FUNCTION_BLOCK FB_VeggiePizza EXTENDS FB_Pizza
VAR_INPUT
END_VAR
VAR_OUTPUT
END_VAR
VAR
END_VAR

METHOD addCheese
VAR_INPUT
END_VAR
ADSLOGSTR( msgCtrlMask := ADSLOG_MSGTYPE_WARN,
        	msgFmtStr := 'Adding Mozzarella Cheese...', '');
END_METHOD

METHOD addMeat
VAR_INPUT
END_VAR
// Nothing here because it's not used
// Normally these Meat, Cheese, and Veg would be an Abstract Method
END_METHOD

METHOD addVegetables : BOOL
VAR_INPUT
END_VAR
ADSLOGSTR( msgCtrlMask := ADSLOG_MSGTYPE_WARN,
        	msgFmtStr := 'Adding Veggies...', '');
END_METHOD

METHOD customerWantsCheese : BOOL
VAR_INPUT
END_VAR
// Cheese Hook
customerWantsCheese := TRUE;
END_METHOD

METHOD customerWantsVegetables : BOOL
VAR_INPUT
END_VAR
// Veggie Hook
customerWantsVegetables := TRUE;
END_METHOD

END_FUNCTION_BLOCK

(* stored: Version 1.1.0.1, ProductVersion 3.1.4024.12
   POU FB_VeggiePizza: Id {dadc269c-d04f-4b7c-b2cb-9fc6e6bef60e}, SpecialFunc None
   Method addCheese: Id {ae4a65a9-b1e9-4f1f-8552-6ec3a26465e1}
   Method addMeat: Id {7d0343f8-6c59-4230-84e0-12aa344593b6}
   Method addVegetables: Id {49fee86e-d8b2-46f4-b43c-2344252176db}
   Method customerWantsCheese: Id {9406d187-e56d-45a7-9bcb-c056c16a05c3}
   Method customerWantsVegetables: Id {c9bacecd-a564-481d-8439-98ba92af03bb} *)
